TYPE ST_BoxRobotRecipe :
STRUCT
	wsCaption											:	WSTRING;	//Nazwa stacji	

	stPickOffsetX									:	ST_LrParametr;	//	Offset poz pobierania x 1mm
	stPickOffsetY									:	ST_LrParametr;	//	Offset poz pobierania x 1mm
	stPickOffsetZ									:	ST_LrParametr;	//	Offset poz pobierania x 1mm
	stPickOffsetA									:	ST_LrParametr;	//	Offset poz pobierania x 1 stopeń
	stPickOffsetB									:	ST_LrParametr;	//	Offset poz pobierania x 1 stopeń
	stPickOffsetC									:	ST_LrParametr;	//	Offset poz pobierania x 1 stopeń
	                                                                      	
	stPickAccelecation								:	ST_UdiParametr;	//	Acc in % [1..100]
	stPickDecceleration								:	ST_UdiParametr;	//	Dec in % [1..100]
	stPickOverride									:	ST_UdiParametr;	//	Override in % [1..100]
	stPickColisionDetect							:	ST_UdiParametr; //	Col awoid in %[1..100]
	stPickGripperDelayTime							:	ST_UdiParametr;	//	Czas dojazdu   ms
	stSuckingTimeOn									:	ST_UdiParametr;	//	Czas posysania ms
	stSuckingTimeOff								:	ST_UdiParametr; //	Czas posysania ms
                                                                          	
	stPlaceOffsetX									:	ST_LrParametr;	//	Offset poz odkladania 2 x 1mm
	stPlaceOffsetY									:	ST_LrParametr;	//	Offset poz odkladania 2 x 1mm
	stPlaceOffsetZ									:	ST_LrParametr;	//	Offset poz odkladania 2 x 1mm
	stPlaceOffsetA									:	ST_LrParametr;	//	Offset poz odkladania 2 x 1 stopeń
	stPlaceOffsetB									:	ST_LrParametr;	//	Offset poz odkladania 2 x 1 stopeń
	stPlaceOffsetC									:	ST_LrParametr;	//	Offset poz odkladania 2 x 1 stopeń
                                                                          	
	stPlaceAccelecation								:	ST_UdiParametr;	//	Acc in % [1..100]
	stPlaceDecceleration							:	ST_UdiParametr;	//	Dec in % [1..100]
	stPlaceOverride									:	ST_UdiParametr;	//	Override in % [1..100]
	stPlaceColisionDetect							:	ST_UdiParametr; //	Col awoid in %[1..100]
	stRezerwa1										:	ST_UdiParametr;	//	
	stRezerwa2										:	ST_UdiParametr; //	
	stRezerwa3										:	ST_UdiParametr;	//	
	stGripperTimeClose								:	ST_UdiParametr;	//	Czas skłądania chwytaka
	stGripperTimeOpen								:	ST_UdiParametr;	//	Czas otwierania chwytaka
	                                                                      	
	stPickPreX										:	ST_LrParametr;	//	Odsuniecie przed pozycją pobierania w osi X      
	stPickPreY										:	ST_LrParametr;	//	Odsuniecie przed pozycją pobierania w osi Y      	
	stPickPreZ										:	ST_LrParametr;	//	Odsuniecie przed pozycją pobierania w osi Z      
	stPickAfterX									:	ST_LrParametr;  //	Odsuniecie po pobraniu w osi X                   
	stPickAfterY		                            :	ST_LrParametr;  //	Odsuniecie po pobraniu w osi Y                   
	stPickAfterZ		                            :	ST_LrParametr;  //	Odsuniecie po pobraniu w osi Z                   
	stPlacePreX										:	ST_LrParametr;  //	Odsuniecie przed pozycją odłożenia w osi X       
	stPlacePreY		                                :	ST_LrParametr;  //	Odsuniecie przed pozycją odłożenia w osi Y       
	stPlacePreZ		                                :	ST_LrParametr;  //	Odsuniecie przed pozycją odłożenia w osi Z       
	stPlaceAfterX		                            :	ST_LrParametr;  //	Odsuniecie po odłożenia w osi X                  
	stPlaceAfterY		                            :	ST_LrParametr;  //	Odsuniecie po odłożenia w osi Y                  
	stPlaceAfterZ		                            :	ST_LrParametr;  //	Odsuniecie po odłożenia w osi Z                  
	stBoxPickHeight									:	ST_LrParametr;       
	stBoxWingDown	  	                            :	ST_LrParametr;  //	Dolna długość krawędzi skrzydła kartonu          
	stCurveMotionPositionZ	  	                    :	ST_LrParametr;  //	Wysokość osłon dla dokładnego wkładania
	stCurveDistanceX	                            :	ST_LrParametr;  //	Offset pozycji najeżdzania na balchę prowadzącą X
	stCurveDistanceY								:	ST_LrParametr;  //	Offset pozycji najeżdzania na balchę prowadzącą Y
	stCurveDistanceZ	                            :	ST_LrParametr;  //	Offset pozycji najeżdzania na balchę prowadzącą Z
	stCurveMotionAngleA								:	ST_LrParametr;  //	Kąt zaokrąglenia włozenia kartonu A
	stCurveMotionAngleB                             :	ST_LrParametr;  //	Kąt zaokrąglenia włozenia kartonu B

END_STRUCT
END_TYPE

(* stored: Version 1.1.0.1, ProductVersion 3.1.4026.13, FileIdentifier d309c2628ce791b05752189e1aeb2f20ad9c17cf, FileSignature 6a847bc4fb3c7ca93ce5e355b6043ed9725ea3bb5c012e69847cb9c11cfdbbd8648f77b90bc869515fc068b02702c6a4d8ec0131b32b50e69ea2b67252634349adc6d87b1be518a2bb29cd31dc8d83ab7b3a746ea5dea104d8dcb39ff926696caea66f8f59be55760d5b2bd608614fd86a1913f163f628338419f6ae851f47d0d8fed556970715f334518a1436bf927ebe55af2f9de0bdd43b91c5864dbf78391f23750c4591d77eab50f190e9a92d9e18c00d13676d2eedfa18e1993cc1272221f984524de5b3f28b3933e1be08a16ffa44478c079d22390bc133d264a9dcc073bca5548ca5631a8553138a192c39dfaa6c96c50ae22026492a01d4abbc7670
   DUT ST_BoxRobotRecipe: Id {6e5ffe54-212e-4f1c-a7ce-cc8a2e70663d} *)
